INTERFACE I_Room EXTENDS I_Arg

PROPERTY Active : BOOL
GET
END_GET
END_PROPERTY

METHOD Close
END_METHOD

PROPERTY Id : UDINT
GET
END_GET
END_PROPERTY

PROPERTY IsClosed : BOOL
GET
END_GET
END_PROPERTY

PROPERTY IsOpen : BOOL
GET
END_GET
END_PROPERTY

PROPERTY IsReady : BOOL
GET
END_GET
END_PROPERTY

METHOD Open
END_METHOD

PROPERTY Timeout : TIME
GET
END_GET
END_PROPERTY

METHOD TriggerFault
VAR_INPUT
	sErrorText		: Str;
END_VAR
END_METHOD

END_INTERFACE

(* stored: Version 1.1.0.1
   Itf I_Room: Id {76a64c62-873b-4b19-9f71-81cd9ae5bd4a}
   Property Active: Id {5180e7d7-76b6-4027-9c3b-6d66e4b3dcda}
   Get Get: Id {bfc8ec5c-38b4-4ae4-af4d-8483d7a2571a}
   Method Close: Id {58e7653f-e1ac-4385-b729-fcc12c30b43f}
   Property Id: Id {f4e2640b-d8af-47d9-82c8-6c5680ee6808}
   Get Get: Id {8d16b22d-5201-4bcd-a435-844623fe0306}
   Property IsClosed: Id {53d44817-54c5-4213-9c59-bed5c2800bbd}
   Get Get: Id {599e20a8-f14b-4911-9121-56f115edd3b3}
   Property IsOpen: Id {a80fed6d-ffd6-4cb9-9946-9a19a16beace}
   Get Get: Id {4a82a473-e1f4-4f1b-bffb-3644abf6cfaf}
   Property IsReady: Id {50c3e0ec-167d-4787-96ca-fe310c4f9f97}
   Get Get: Id {778bad79-aa64-4466-94de-baac6b08b962}
   Method Open: Id {5a95de94-7557-4aa0-b324-b5fe346d2f7b}
   Property Timeout: Id {823ffe10-9a79-49a6-bd9e-fd2178fd5d66}
   Get Get: Id {f1995043-f163-4a8a-bc8d-7b4ff2103cd7}
   Method TriggerFault: Id {1713fcd6-0c02-4d9f-a5f9-4c020ec3bb1f} *)
